{attribute 'linkalways'} 
{attribute 'no_explicit_call' := 'This FB is a CLASS and must be accessed using methods or properties'}
{attribute 'enable_dynamic_creation'}
FUNCTION_BLOCK DictionaryTreeNode EXTENDS Disposable IMPLEMENTS I_DictionaryTreeNode
VAR
	_key : T_MAXSTRING;
	pBuffer : POINTER TO BYTE;
	bufferSize : UDINT;
    _height : DINT;
    _left : I_DictionaryTreeNode;
    _right : I_DictionaryTreeNode;
END_VAR

METHOD PRIVATE CopyBufferToDestination
VAR_INPUT
	DestinationAddress : PVOID;
END_VAR
MEMCPY(DestinationAddress, pBuffer, bufferSize);
END_METHOD

METHOD PRIVATE CopySourceToBuffer
VAR_INPUT
	SourceAddress : PVOID;
END_VAR
MEMCPY(pBuffer, SourceAddress, bufferSize);
END_METHOD

METHOD PRIVATE CreateBuffer
VAR_INPUT
	SizeInBytes : UDINT;
END_VAR
bufferSize := SizeInBytes;
pBuffer := __NEW(BYTE, SizeInBytes);
END_METHOD

PROPERTY PUBLIC DataSize : UDINT
GET
DataSize := bufferSize;
END_GET
END_PROPERTY

METHOD PRIVATE DestroyBuffer
VAR_INPUT
END_VAR
IF pBuffer = 0 THEN
	RETURN;
END_IF

__DELETE(pBuffer);
bufferSize := 0;
END_METHOD

METHOD PUBLIC Equals : BOOL
VAR_INPUT
	Symbol : ANY;
END_VAR
IF pBuffer = 0 THEN
	RETURN;
END_IF

IF bufferSize <> DINT_TO_UDINT(symbol.diSize) THEN
	RETURN;
END_IF

Equals := MEMCMP(Symbol.pValue, pBuffer, bufferSize) = 0;
END_METHOD

METHOD FB_exit : BOOL
VAR_INPUT
	bInCopyCode : BOOL; // if TRUE, the exit method is called for exiting an instance that is copied afterwards (online change).
END_VAR
IF bInCopyCode THEN
	RETURN;
END_IF

DestroyBuffer();
END_METHOD

PROPERTY PUBLIC Height : DINT
GET
Height := _height;
END_GET
SET // PUBLIC
_height := Height;
END_SET
END_PROPERTY

METHOD Initialize
VAR_INPUT
	Key : T_MAXSTRING;
	Value : ANY;
END_VAR
_key := Key;

IF pBuffer <> 0 THEN
	DestroyBuffer();
END_IF

CreateBuffer(DINT_TO_UDINT(Value.diSize));
CopySourceToBuffer(Value.pValue);
END_METHOD

PROPERTY PUBLIC Key : T_MAXSTRING
GET
Key := _key;
END_GET
END_PROPERTY

PROPERTY PUBLIC Left : I_DictionaryTreeNode
GET
Left := _left;
END_GET
SET
_left := Left;
END_SET
END_PROPERTY

PROPERTY PUBLIC Right : I_DictionaryTreeNode
GET
Right := _right;
END_GET
SET
_right := Right;
END_SET
END_PROPERTY

METHOD TryGet : BOOL
VAR_INPUT
	Destination	: ANY;
END_VAR
TryGet := TryGetTo(Destination.pValue, DINT_TO_UDINT(Destination.diSize));
END_METHOD

METHOD TryGetTo : BOOL
VAR_INPUT
	DestinationAddress : PVOID;
	DestinationSize : UDINT;
END_VAR
IF pBuffer = 0 THEN
	RETURN;
END_IF

IF bufferSize <> DestinationSize THEN
	RETURN;
END_IF

CopyBufferToDestination(DestinationAddress);
TryGetTo := TRUE;
END_METHOD

END_FUNCTION_BLOCK

(* stored: Version 1.1.0.1, ProductVersion 3.1.4024.12
   POU DictionaryTreeNode: Id {f814d24b-144d-4d3c-90bc-13c52ba890ae}, SpecialFunc None
   Folder Destructor: Id {78526f89-48f1-436e-9832-12e9ed8b469e}
   Folder Private: Id {8d481354-6053-40a3-b6f8-e65f747ac3db}
   Method CopyBufferToDestination: Id {f1c92538-a371-4a93-8465-74398204a812}
   Method CopySourceToBuffer: Id {c160ccd2-a837-45fc-b9b6-86421ded89c3}
   Method CreateBuffer: Id {f40ae281-3b0e-446b-9d48-e81c6fd1bfc4}
   Property DataSize: Id {40dd125d-f1d3-4009-ba0a-51ce85c51735}
   Get Get: Id {89a5ce5a-4e7e-43fe-ab41-59195951ac65}
   Method DestroyBuffer: Id {465cd18c-2bc6-4e44-9ca2-886cbba69f41}
   Method Equals: Id {8bf6e19a-5459-4b03-9f44-9e6adbb801b7}
   Method FB_exit: Id {4892f69d-02d1-4b08-aeb8-a4d64d04e10a}
   Property Height: Id {537a2615-9865-4110-a955-9ed8dc640b6c}
   Get Get: Id {a9921c6b-ddbe-4426-8ba4-0fcf447142ed}
   Set Set: Id {1906fbf1-f80d-4361-8079-7aa297738b01}
   Method Initialize: Id {cd8e08b7-7703-46a4-b8ab-44543cf0a164}
   Property Key: Id {ec56e455-80e8-48e4-8ca2-8341fce7f467}
   Get Get: Id {1c175802-131e-4874-b3f2-1522775aaf15}
   Property Left: Id {cdb84292-ecaf-424d-934b-a88faaedf26d}
   Get Get: Id {f648b350-562b-4adc-9698-14878f00345a}
   Set Set: Id {6523ddb3-c975-43ca-96e7-22ff343aeb04}
   Property Right: Id {0eeff03f-7821-48fe-8897-9945f59363f5}
   Get Get: Id {496229f8-c9ab-4df6-9d59-37c887fa16ae}
   Set Set: Id {5e907fa5-75f5-4d37-88ab-0e5b572da295}
   Method TryGet: Id {89c16e15-b563-4229-86c3-0bd48b463b8d}
   Method TryGetTo: Id {502b73dd-cd36-4d33-912b-fcfb6a460d07} *)
